# EPICS substitutions: LKSH336/LKSH336-IOC-01App/Db/lakeshore336.substitutions
file $(LKSH336)/db/lakeshore336.template
{
pattern {P, PORT, ADDR, TEMPSCAN, SCAN}
	{"\$(P)", "\$(PORT)", 0, 1, 5}
}

file $(LKSH336)/db/lakeshore336_SIM.template
{
pattern {P}
	{"\$(P)"}
}
